# EPICS autosave request: apps/chicaneApp/Db/chicane_settings.req
$(P):energy
$(P):iCalcPS
$(P):iCalcMT
$(P):tHoldMax
$(P):iDelta
